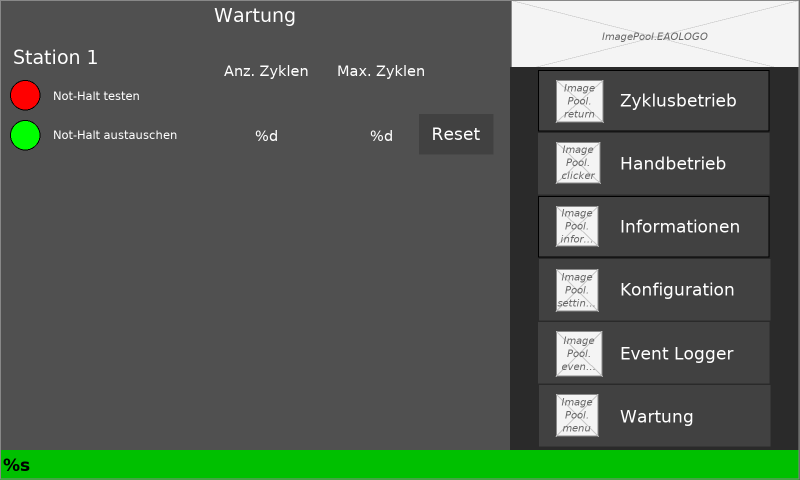
VISUALIZATION Wartung  // 800x480
    Image (511,0 288x73), image: ImagePool.EAOLOGO
    Rectangle (510,67 289x412)
    Textfield (155,1 200x29), "Wartung"
    Rectangle (0,450 799x30), "%s", text variable: MAIN.HMI.sStatus, colour variable: MAIN.HMI.nColorInfoBalken
        p3450524324: MAIN.HMI.nColorInfoBalken
    Rectangle (538,70 231x61)
        OnMouseClick: change screen: Zyklusbetrieb
    Textfield (617,70 153x61), "Zyklusbetrieb"
        OnMouseClick: change screen: Zyklusbetrieb
    Rectangle (538,133 231x61)
        OnMouseClick: change screen: Handbetrieb
    Textfield (617,133 153x61), "Handbetrieb"
        OnMouseClick: change screen: Handbetrieb
    Image (556,142 44x41), image: ImagePool.clicker
        OnMouseClick: change screen: Handbetrieb
    Image (556,80 47x42), image: ImagePool.return
        OnMouseClick: change screen: Zyklusbetrieb
    Rectangle (538,196 231x61)
        OnMouseClick: change screen: Diagnose
    Textfield (617,196 153x61), "Informationen"
        OnMouseClick: change screen: Diagnose
    Image (556,206 42x40), image: ImagePool.information
        OnMouseClick: change screen: Diagnose
    Rectangle (538,322 231x61)
        OnMouseClick: change screen: EventLogger
    Textfield (617,323 153x61), "Event Logger"
        OnMouseClick: change screen: EventLogger
    Image (556,331 46x45), image: ImagePool.eventLogger
        OnMouseClick: change screen: EventLogger
    Rectangle (539,259 231x61)
        OnMouseClick: change screen: Konfig1
    Textfield (617,259 153x61), "Konfiguration"
        OnMouseClick: change screen: Konfig1
    Image (556,269 42x42), image: ImagePool.settings
        OnMouseDown: change screen: Konfig1
    Rectangle (539,385 231x61)
        OnMouseClick: change screen: Wartung
    Textfield (617,386 153x61), "Wartung"
        OnMouseClick: change screen: Wartung
    Image (556,394 42x42), image: ImagePool.menu
        OnMouseDown: change screen: Wartung
    Textfield (50,80 199x32), "Not-Halt testen"
    Textfield (50,120 204x30), "Not-Halt austauschen"
    Ellipse (10,80 30x30), colour toggle: MAIN.fbSt1.bNotHaltTestIO
    Ellipse (10,120 30x30), colour toggle: MAIN.fbSt1.bWarnungNothalt
    Textfield (367,120 78x32), "%d", text variable: Parameter.cMaxZyklNotHalt
    Textfield (252,120 78x32), "%d", text variable: MAIN.fbSt1.nZaehlerNotHalt
    Textfield (221,55 105x32), "Anz. Zyklen"
    Textfield (334,55 105x32), "Max. Zyklen"
    RoundedRectangle (419,114 74x40), "Reset", invisible if: NOT MAIN.fbSt1.bWarnungNothalt
        OnMouseClick: execute { MAIN.fbSt1.bBtnResetWarnNothalt := TRUE; }
    Textfield (10,43 200x29), "Station 1"
END_VISUALIZATION

(* stored: Version 1.1.0.1, ProductVersion 3.1.4024.12
   Visu Wartung: Id {f24f2c9b-f586-46e4-b8da-bc4e8577d3cb} *)
